TYPE ST_STATUS_ROT :
STRUCT
		bPhaseOK:BOOL:=FALSE;
END_STRUCT
END_TYPE

(* stored: Version 1.1.0.1, ProductVersion 3.1.4024.6
   DUT ST_STATUS_ROT: Id {6c493b2f-cb6a-4fc1-849c-d8e5ead15e5e} *)
